(* 
:Description: This function block is used represent basic axis controled by standard PLCopen motion function blocks.
*)
FUNCTION_BLOCK FB_AxisServo EXTENDS FB_UniversalAxis
VAR
	(* MC_Home *)
	eHomingMode		: MC_HomingMode;		(*  *)
	stHomingOptions	: ST_HomingOptions;		(*  *)
	fbMcHome		: MC_Home;				(*  *)
	
	(* Home switch cam *)
	piHomeSwitch	: FB_DigitalInput;		(*  *)
END_VAR
(*
Version history:

+-------------+------------+----------------+----------+------------------------------------------+
|Date         | Version    | created under  | Author   | Remark                                   |
+=============+============+================+==========+==========================================+
|2021-11      | 1.0.0.0    | V3.1.4024.22   | ADBO     | Function block created                   |
+-------------+------------+----------------+----------+------------------------------------------+

*)

(* Run home switch FB *)
piHomeSwitch();

(* Run parent implementation *)
SUPER^();

PROPERTY HomingMode : MC_HomingMode
GET
HomingMode := eHomingMode;
END_GET
SET
eHomingMode := HomingMode;
END_SET
END_PROPERTY

PROPERTY HomingOptions : ST_HomingOptions
GET
HomingOptions := stHomingOptions;
END_GET
SET
stHomingOptions := HomingOptions;
END_SET
END_PROPERTY

METHOD MR_FirstCycle
VAR_INPUT
	sName 				: STRING; 	(* Axis object name *)
	sMeasurementUnits	: STRING;	(* Measurement units used by axis *)
	bModulo				: BOOL;		(* Axis is periodic *)
END_VAR
SUPER^.MR_FirstCycle(sName:=sName, sMeasurementUnits := sMeasurementUnits, bModulo := bModulo);
piHomeSwitch.MR_FirstCycle(CONCAT(THIS^.sName,', home switch'), sModuleType := piHomeSwitch.ModuleType, sPortID := piHomeSwitch.PortID);
END_METHOD

(* 
Copyrights	: Sonion Industrialization - Control Systems Desing Department
Author		: Adrian Bogdzia - based on MEMS universal libraries
Date		: 11/2021
Description : This function block is used represent basic axis
*)
METHOD PROTECTED MS_Aborting
VAR_INPUT
END_VAR
fbMcHome(Axis := stAxisRef, Execute := FALSE);

SUPER^.MS_Aborting();
END_METHOD

(* 
Copyrights	: Sonion Industrialization - Control Systems Desing Department
Author		: Adrian Bogdzia - based on MEMS universal libraries
Date		: 11/2021
Description : This function block is used represent basic axis
*)
METHOD PROTECTED MS_Halt
VAR_INPUT
END_VAR
(* Reset MC_Home *)
fbMcHome(Axis := stAxisRef, Execute := FALSE);

(* Run parent halt state *)
SUPER^.MS_Halt();
END_METHOD

(* 
Copyrights	: Sonion Industrialization - Control Systems Desing Department
Author		: Adrian Bogdzia - based on MEMS universal libraries
Date		: 11/2021
Description : This function block is used represent basic axis
*)
METHOD PROTECTED MS_Home
VAR_INPUT
END_VAR
fbMcHome(	Axis 			:= stAxisRef,
			Execute 		:= TRUE,
			Position 		:= lrHomePosition,
			HomingMode		:= eHomingMode,
			BufferMode		:= eBufferMode,
			Options			:= stHomingOptions,
			bCalibrationCam := piHomeSwitch.In);
	
IF fbMcHome.Error THEN
	bError := TRUE;
	iErrorID := fbMcHome.ErrorID;
	fbMcHome( Axis := stAxisRef, Execute := FALSE);
	fbAlarmHome.ipArguments.Clear().AddUDInt(iErrorID);	
	fbAlarmHome.Raise(0);
	
ELSIF fbMcHome.Done THEN
	eAxisState := AXIS_HOME_DONE;
		
END_IF
END_METHOD

(* 
Copyrights	: Sonion Industrialization - Control Systems Desing Department
Author		: Adrian Bogdzia - based on MEMS universal libraries
Date		: 11/2021
Description : This function block is used represent basic axis
*)
METHOD PROTECTED MS_HomeDone
VAR_INPUT
END_VAR
fbMcHome(Axis := stAxisRef, Execute := FALSE);

IF NOT bHome AND NOT fbMcHome.Busy THEN
	eAxisState := AXIS_IDLE;
	
END_IF
END_METHOD

(* 
Copyrights	: Sonion Industrialization - Control Systems Desing Department
Author		: Adrian Bogdzia - based on MEMS universal libraries
Date		: 11/2021
Description : This function block is used represent basic axis
*)
METHOD PROTECTED MS_Reset
VAR_INPUT
END_VAR
(* Reset MC_Home*)
fbMcHome( Axis := stAxisRef, Execute := FALSE);

(* Run parent reset procedure*)
IF NOT fbMcHome.Busy THEN
	SUPER^.MS_Reset();
	
END_IF
END_METHOD

(* 
Copyrights	: Precision System Engineering - Control Systems Desing Department
Author		: Adrian Bogdzia - based on MEMS universal libraries
Date		: 11/2021
Description : This function block is used represent basic axis
*)
METHOD PROTECTED MS_Stop
VAR_INPUT
END_VAR
(* Reset MC_Home *)
fbMcHome(Axis := stAxisRef, Execute := FALSE);

(* Run parent stop state *)
SUPER^.MS_Stop();
END_METHOD

PROPERTY ref_HomeSwitch : REFERENCE TO FB_DigitalInput
GET
ref_HomeSwitch REF= piHomeSwitch;
END_GET
END_PROPERTY

END_FUNCTION_BLOCK

(* stored: Version 1.1.0.1, ProductVersion 3.1.4024.9
   POU FB_AxisServo: Id {6589cba5-148f-47a8-a127-24cca4ed91b7}, SpecialFunc None
   Folder FirstCycle: Id {275be946-a97f-4cd6-ac88-a77d288adf62}
   Folder Properties: Id {68a0a49a-42fa-436b-9f8e-cefc53d48124}
   Folder Parameters: Id {57e6479d-26fb-4cfc-9593-a832538be85c}
   Folder References: Id {868e607b-db85-4cbf-8453-87b1960811c9}
   Folder StateMachine: Id {3818c0d8-5ceb-45e0-97b0-bce4798f0584}
   Property HomingMode: Id {17642853-32ab-43a0-bc98-a79e76ac9a69}
   Get Get: Id {b34f8398-ee30-4bbe-93b2-416d9fb66a66}
   Set Set: Id {0edc2f2b-ffb0-4c1d-b0a9-72286a36b913}
   Property HomingOptions: Id {bd4f7f18-29dc-4871-afdb-41403620f3b1}
   Get Get: Id {bdbfc0e9-9201-4720-b28a-72ccdc9188d7}
   Set Set: Id {d9b8db89-2e0b-4cea-b6df-9b8d2e036a23}
   Method MR_FirstCycle: Id {a6240142-a4cb-4304-bf27-57ef3e4a0fd1}
   Method MS_Aborting: Id {f2b50b86-35b5-4226-9eba-2c1b885215f9}
   Method MS_Halt: Id {7627eb40-8a5d-480b-a0d3-149c62505a5a}
   Method MS_Home: Id {c2e538ba-b38a-4fd5-887f-aed7bd7f7379}
   Method MS_HomeDone: Id {5fbc7ac4-b8b3-45ff-a136-276ceff471dd}
   Method MS_Reset: Id {d9bee0f3-2ce6-4521-a42e-e3c3211d68bc}
   Method MS_Stop: Id {7feef091-de7d-4245-bd41-05966da1c68d}
   Property ref_HomeSwitch: Id {53c50a6b-bef8-43c8-a00e-41f6a7da6cc3}
   Get Get: Id {897e0756-9bf6-4477-826c-73e327ad084b} *)
